// Mitsubishi GX Works2 project: 0709계산기   PLC: Q02/Q02H

PROGRAM MAIN
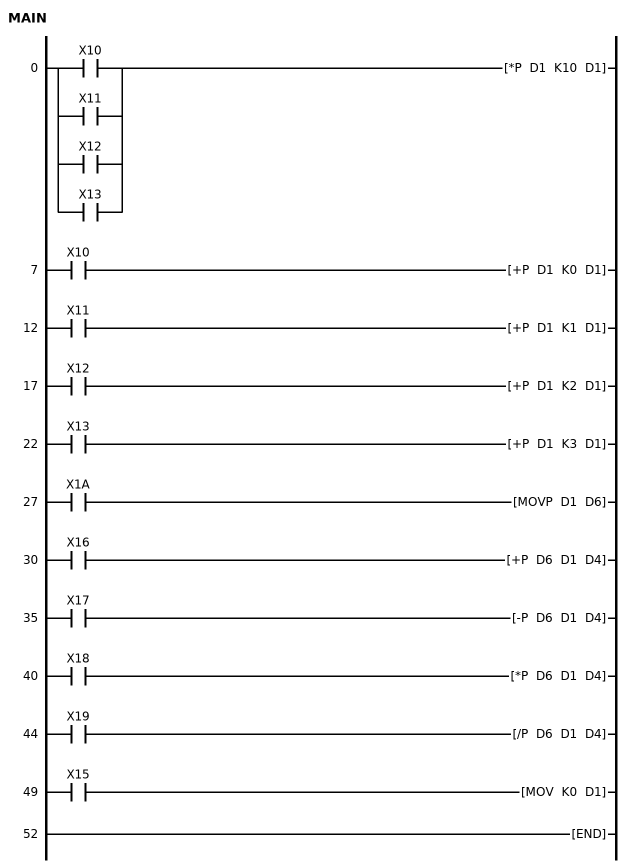
0     LD      X10
      OR      X11
      OR      X12
      OR      X13
      *P      D1 K10 D1
7     LD      X10
      +P      D1 K0 D1
12    LD      X11
      +P      D1 K1 D1
17    LD      X12
      +P      D1 K2 D1
22    LD      X13
      +P      D1 K3 D1
27    LD      X1A
      MOVP    D1 D6
30    LD      X16
      +P      D6 D1 D4
35    LD      X17
      -P      D6 D1 D4
40    LD      X18
      *P      D6 D1 D4
44    LD      X19
      /P      D6 D1 D4
49    LD      X15
      MOV     K0 D1
52    END
END_PROGRAM
